KUKA KRL program: vw_hlf_usr_s.src, vw_hlf_usr_s.dat

--- vw_hlf_usr_s.src ---
&ACCESS RVEO
&REL 6
&COMMENT KS24.24.000_VW
&PARAM TPVW_VERSION = 8.1.8
&PARAM DISKPATH = VW_User / Applikation / VW_Grei_Fehl
DEF vw_hlf_usr_s( )
   ;
   ;*-----------------------------------------------------*
   ;* Erstellt am:                                        *
   ;* 2017.11.03                                          *
   ;*------------------------------------------------------
   ;
END
;
;FOLD INIT Handl_Fehl
GLOBAL DEF HLF_INIT( )
INT i
;;
;
END
;ENDFOLD
;
;-----------------------------------------------------------
;FOLD SAW Handl_Fehl
GLOBAL DEF HLF_SAW( )
INT i
;
;
END
;ENDFOLD
;
;-----------------------------------------------------------
;FOLD RESET Handl_Fehl
GLOBAL DEF HLF_RESET( )
INT i
;
;
END
;ENDFOLD
;
;-----------------------------------------------------------
;FOLD CANCEL Handl_Fehl
GLOBAL DEF HLF_CANCEL( )
INT i
;
;
END
;ENDFOLD
;
;-----------------------------------------------------------
;FOLD LOOP Handl_Fehl
GLOBAL DEF HLF_LOOP( )
INT i, j, k
BOOL R_POS_ABFRA
BOOL V_POS_ABFRA


FOR i = 1 TO 22
;Schleifentest
    CONTINUE
	IF ($OUT[15]==TRUE) OR ($IN[15]==TRUE) THEN  ; Bei Grundstellung alle Greifer deaktivieren
	;Fehlermedungen OFF
	  HLF_SPGR_AKT[i]=FALSE
	  HLF_F_SPANNZ=0
	  HLF_A_BIS_H=0
      FEHLER_SPG=0
      FEHLER_GRU=0
	  FEHLER_TKO=0
	  HLF_KLEIN_A_B=0
	  CONTINUE
	  $OUT[HLF_BGE_V_R]=FALSE
	  CONTINUE
      $OUT[HLF_BGE_SP_A]=FALSE
		IF i <=15 THEN
	       HLF_BGEKONT[i]=FALSE
		ENDIF
	ENDIF
	;------------------------------------------------------------------
	k=1
	CONTINUE
    IF (HLF_SPGR_AKT[i]==TRUE) AND ($IN[15]==FALSE)  AND (HLF_OPT_SPS>=127) AND (HLF_OPT_SPS<=257) THEN  ;Spanngruppe aktiv
        ;-----Spanngruppe ist geschlossen--------------
    	IF (HLF_SPGR_AUF[I]==FALSE) THEN ; Spanngruppe ist geschlossen
	     FOR j = 1 TO (HLF_ANZ_SGRUP[i])  ; 2
		 ;----------Wechsel zwischen Abfrageposition
			IF (J==1) THEN
				R_POS_ABFRA=TRUE
				IF (HLF_ERSBIT_R[i]==TRUE) THEN  ; Erstes Bit ist R Pos
					R_POS_ABFRA=FALSE
				ENDIF
			ELSE
				IF (R_POS_ABFRA==FALSE) THEN
					R_POS_ABFRA=TRUE
				ELSE
					R_POS_ABFRA=FALSE
				ENDIF
			ENDIF
            ;-------ENDE---Wechsel zwischen Abfrageposition
          ;-----Kontrolle Spanngruppe--------------
			CONTINUE
         IF ( (HLF_ST_ADR_SG[i]+(j-1))<1) OR  ((HLF_ST_ADR_SG[i]+(j-1))> 4096) THEN
				HLF_ST_ADR_SG[i]=4070
			ENDIF
		    IF ($IN[(HLF_ST_ADR_SG[i]+(j-1))]<>R_POS_ABFRA) THEN ;; Kontrolle Position NIO
                IF (FEHLER_SPG<1) THEN
					;; FEHLERAUSGABE
					HLF_F_SPANNZ=i
					HLF_A_BIS_H=(j+1)/2
					HLF_KLEIN_A_B=0
					FEHLER_SPG=i
					FEHLER_GRU=j
					CONTINUE
					$OUT[HLF_BGE_V_R]= TRUE
					IF (i<17) THEN   ; Ausgabe Bit 11 Spanngruppe = True
						CONTINUE
					   $OUT[HLF_BGE_SP_A]=TRUE
					ELSE  ; Ausgabe Bit 11 Sauger = False
						CONTINUE
					   $OUT[HLF_BGE_SP_A]=FALSE
					   HLF_A_BIS_H=0
					ENDIF
				ENDIF
			ELSE
				IF (FEHLER_SPG>0) THEN  ; Fehler loeschen
					IF (FEHLER_SPG==i) AND (FEHLER_GRU==j) THEN
						HLF_F_SPANNZ=0
						HLF_A_BIS_H=0
						FEHLER_SPG=0
						FEHLER_GRU=0
						CONTINUE
						$OUT[HLF_BGE_V_R]=FALSE
						CONTINUE
						$OUT[HLF_BGE_SP_A]=FALSE
					ENDIF
				ENDIF
			ENDIF

		 ENDFOR
		 ;---ENDE--Spanngruppe ist geschlossen--------------
	   ELSE
	        ;---Start--Spanngruppe ist offen--------------
		FOR j = 1 TO (HLF_ANZ_SGRUP[i])
		    ;----------Wechsel zwischen Abfrageposition
			IF (J==1) THEN
				V_POS_ABFRA=FALSE
				IF (HLF_ERSBIT_R[i]==TRUE) THEN  ; Erstes Bit ist R Pos
					V_POS_ABFRA=TRUE
				ENDIF
			ELSE
				IF (V_POS_ABFRA==FALSE) THEN
					V_POS_ABFRA=TRUE
				ELSE
					V_POS_ABFRA=FALSE
				ENDIF
			ENDIF
            ;-------ENDE---Wechsel zwischen Abfrageposition
          ;-----Kontrolle Spanngruppe--------------

			CONTINUE
		    IF ($IN[(HLF_ST_ADR_SG[i]+(j-1))]<>V_POS_ABFRA) THEN ;; Kontrolle Position NIO
                IF (FEHLER_SPG<1) THEN
					;; FEHLERAUSGABE
					HLF_F_SPANNZ=i
					HLF_A_BIS_H=(j+1)/2
					HLF_KLEIN_A_B=0
					FEHLER_SPG=i
					FEHLER_GRU=j
					CONTINUE
					$OUT[HLF_BGE_V_R]= FALSE
					IF (i<17) THEN   ; Ausgabe Bit 11 Spanngruppe = True
						CONTINUE
					   $OUT[HLF_BGE_SP_A]=TRUE
					ELSE  ; Ausgabe Bit 11 Sauger = False
					   CONTINUE
					   $OUT[HLF_BGE_SP_A]=FALSE
					   HLF_A_BIS_H=0
					ENDIF
				ENDIF
			ELSE
				IF (FEHLER_SPG>0) THEN  ; Fehler loeschen
					IF (FEHLER_SPG==i) AND (FEHLER_GRU==j) THEN
						HLF_F_SPANNZ=0
						HLF_A_BIS_H=0
						FEHLER_SPG=0
						FEHLER_GRU=0
						CONTINUE
						$OUT[HLF_BGE_V_R]=FALSE
						CONTINUE
						$OUT[HLF_BGE_SP_A]=FALSE
					ENDIF
				ENDIF
			ENDIF

		 ENDFOR

			;---ENDE--Spanngruppe ist geschlossen--------------
	   ENDIF
    ELSE
	  IF (HLF_SPGR_AKT[i]==FALSE) AND (FEHLER_SPG==i) THEN
   	     HLF_F_SPANNZ=0
	     HLF_A_BIS_H=0
         FEHLER_SPG=0
         FEHLER_GRU=0
	     CONTINUE
		 $OUT[HLF_BGE_V_R]=FALSE
         CONTINUE
		 $OUT[HLF_BGE_SP_A]=FALSE
	  ENDIF

	ENDIF


;------------Teilkontrolle----------------

	CONTINUE
	If (i<=15) AND (HLF_F_SPANNZ<=0) AND ($IN[15]==FALSE) THEN ; Teilkontrollen
		IF (HLF_BGEKONT[i]==FALSE) AND (FEHLER_TKO==i) THEN ;FEHLER Ruecksetzen wenn nicht aktiv
			HLF_A_BIS_H=0
			FEHLER_TKO=0
			HLF_KLEIN_A_B=0
		ENDIF
		IF (HLF_BGEBITA[i]<1) OR (HLF_BGEBITA[i]>4096) THEN ; Fehlerabfang Abfrage Eingabe
         HLF_BGEBITA[i]=4070
		ENDIF
		IF (HLF_BGEBITB[i]<1) OR (HLF_BGEBITB[i]>4096) THEN  ; Fehlerabfang Abfrage Eingabe
         HLF_BGEBITB[i]=4070
		ENDIF
		IF (HLF_BGEKONT[i]==TRUE) AND ((FEHLER_TKO==i) OR (FEHLER_TKO<=0)) THEN   ;Bauteilkontrolle aktiv und (aktueller Fehler oder kein Fehler)
			IF (HLF_BGETEILV[i]==TRUE) THEN  ; Teilkontrolle Teil ist vorhanden
				CONTINUE
				IF (HLF_BGEMITAB[i]==TRUE) THEN  ;Mit klein A und B
					IF ($IN[(HLF_BGEBITA[i])]==TRUE) AND ($IN[(HLF_BGEBITB[i])]==TRUE) THEN ;; Bauteilkontrolle klein A Nicht vorhanden
						IF (FEHLER_TKO==i)  THEN ; Rücksetzen Fehler
							HLF_A_BIS_H=0
							FEHLER_TKO=0
							HLF_KLEIN_A_B=0
						ENDIF
					ELSE  ; FEHLERAUSGABE
						HLF_A_BIS_H=i
						FEHLER_TKO=i
						IF ($IN[(HLF_BGEBITA[i])]==FALSE) THEN
							HLF_KLEIN_A_B=1
						ELSE
							HLF_KLEIN_A_B=2
						ENDIF
					ENDIF

				ELSE   ; Ohne klein A und B
					IF ($IN[(HLF_BGEBITA[i])]==TRUE) THEN ;; Bauteilkontrolle klein A auf vorhanden
						IF (FEHLER_TKO==i)  THEN ; Rücksetzen Fehler
							HLF_A_BIS_H=0
							FEHLER_TKO=0
							HLF_KLEIN_A_B=0
						ENDIF
					ELSE  ; FEHLERAUSGABE
						HLF_A_BIS_H=i
						FEHLER_TKO=i
						HLF_KLEIN_A_B=0
					ENDIF
				ENDIF
			ELSE  ; Teilkontrolle Teil ist NICHT vorhanden

;------------     Auswertung Teilkontrolle KEIN Teil vorhanden
				IF (HLF_BGEMITAB[i]==TRUE) THEN  ;Mit klein A und B
					IF ($IN[(HLF_BGEBITA[i])]==FALSE) AND ($IN[(HLF_BGEBITB[i])]==FALSE) THEN ;; Bauteilkontrolle klein A Nicht vorhanden
						IF (FEHLER_TKO==i)  THEN ; Rücksetzen Fehler
							HLF_A_BIS_H=0
							FEHLER_TKO=0
							HLF_KLEIN_A_B=0
						ENDIF
					ELSE  ; FEHLERAUSGABE
						HLF_A_BIS_H=i
						FEHLER_TKO=i
						IF ($IN[(HLF_BGEBITA[i])]==TRUE) THEN
							HLF_KLEIN_A_B=1
						ELSE
							HLF_KLEIN_A_B=2
						ENDIF
					ENDIF

				ELSE   ; Ohne klein A und B

					IF ($IN[(HLF_BGEBITA[i])]==FALSE) THEN ;; Bauteilkontrolle klein A Nicht vorhanden
						IF (FEHLER_TKO==i)  THEN ; Rücksetzen Fehler
							HLF_A_BIS_H=0
							FEHLER_TKO=0
							HLF_KLEIN_A_B=0
						ENDIF
					ELSE  ; FEHLERAUSGABE
						HLF_A_BIS_H=i
						FEHLER_TKO=i
						HLF_KLEIN_A_B=0
					ENDIF

				ENDIF


			ENDIF ; Teilkontrolle Teil ist vorhanden ENDE
		ENDIF  ; Bauteilkontrolle ENDE
		;;;;; KLEIB b
    ;  ---------------------------

	ENDIF

	IF (HLF_OPT_SPS>127) THEN
		CONTINUE
		HLF_BIN5_AUS((HLF_OPT_SPS), HLF_F_SPANNZ) ; Ausgabe Spannzylinder
		CONTINUE
		HLF_BIN4_AUS((HLF_OPT_SPS+5), HLF_A_BIS_H) ; Ausgabe Teilkontrolle
		CONTINUE
		HLF_BIN2_AUS((HLF_OPT_SPS+11), HLF_KLEIN_A_B) ; Ausgabe Klein A_B
	ENDIF
ENDFOR
;
END
;ENDFOLD

;FOLD Werteausgabe 4 BIT
DEF HLF_BIN4_AUS(HLF_STARTADD :IN, HLF_WERT :IN)
INT HLF_STARTADD, HLF_WERT
IF (HLF_STARTADD>0) AND (HLF_STARTADD<500) AND (HLF_WERT<17) AND (HLF_WERT>=0) THEN

	IF (HLF_WERT>=8) THEN
		HLF_WERT = (HLF_WERT-8)
		CONTINUE
		$OUT[HLF_STARTADD+3]=TRUE
	ELSE
		CONTINUE
		$OUT[HLF_STARTADD+3]=FALSE
	ENDIF

	IF (HLF_WERT>=4) THEN
		HLF_WERT = (HLF_WERT-4)
		CONTINUE
		$OUT[(HLF_STARTADD+2)]=TRUE
	ELSE
		CONTINUE
		$OUT[(HLF_STARTADD+2)]=FALSE
	ENDIF

	IF (HLF_WERT>=2) THEN
		HLF_WERT = (HLF_WERT-2)
		CONTINUE
		$OUT[(HLF_STARTADD+1)]=TRUE
	ELSE
		CONTINUE
		$OUT[(HLF_STARTADD+1)]=FALSE
	ENDIF

		IF (HLF_WERT>=1) THEN
		HLF_WERT = (HLF_WERT-1)
		CONTINUE
		$OUT[(HLF_STARTADD)]=TRUE
	ELSE
		CONTINUE
		$OUT[(HLF_STARTADD)]=FALSE
	ENDIF


ENDIF

END
;ENDFOLD

;FOLD Werteausgabe 5 BIT
DEF HLF_BIN5_AUS(HLF_STARTADD :IN, HLF_WERT :IN)
INT HLF_STARTADD, HLF_WERT
IF (HLF_STARTADD>0) AND (HLF_STARTADD<500) AND (HLF_WERT<33) AND (HLF_WERT>=0) AND (HLF_OPT_SPS>127) THEN

	IF (HLF_WERT>=16) THEN
		HLF_WERT = (HLF_WERT-16)
		CONTINUE
		$OUT[HLF_STARTADD+4]=TRUE
	ELSE
		CONTINUE
		$OUT[HLF_STARTADD+4]=FALSE
	ENDIF

	IF (HLF_WERT>=8) THEN
		HLF_WERT = (HLF_WERT-8)
		CONTINUE
		$OUT[HLF_STARTADD+3]=TRUE
	ELSE
		CONTINUE
		$OUT[HLF_STARTADD+3]=FALSE
	ENDIF

	IF (HLF_WERT>=4) THEN
		HLF_WERT = (HLF_WERT-4)
		CONTINUE
		$OUT[(HLF_STARTADD+2)]=TRUE
	ELSE
		CONTINUE
		$OUT[(HLF_STARTADD+2)]=FALSE
	ENDIF

	IF (HLF_WERT>=2) THEN
		HLF_WERT = (HLF_WERT-2)
		CONTINUE
		$OUT[(HLF_STARTADD+1)]=TRUE
	ELSE
		CONTINUE
		$OUT[(HLF_STARTADD+1)]=FALSE
	ENDIF

		IF (HLF_WERT>=1) THEN
		HLF_WERT = (HLF_WERT-1)
		CONTINUE
		$OUT[(HLF_STARTADD)]=TRUE
	ELSE
		CONTINUE
		$OUT[(HLF_STARTADD)]=FALSE
	ENDIF

ENDIF

END
;ENDFOLD

;FOLD Werteausgabe 2 BIT
DEF HLF_BIN2_AUS(HLF_STARTADD :IN, HLF_WERT :IN)
INT HLF_STARTADD, HLF_WERT
IF (HLF_STARTADD>0) AND (HLF_STARTADD<500) AND(HLF_WERT<4) AND (HLF_WERT>=0) AND (HLF_OPT_SPS>127) THEN


	IF (HLF_WERT>=2) THEN
		HLF_WERT = (HLF_WERT-2)
		CONTINUE
		$OUT[(HLF_STARTADD+1)]=TRUE
	ELSE
		CONTINUE
		$OUT[(HLF_STARTADD+1)]=FALSE
	ENDIF

		IF (HLF_WERT>=1) THEN
		HLF_WERT = (HLF_WERT-1)
		CONTINUE
		$OUT[(HLF_STARTADD)]=TRUE
	ELSE
		CONTINUE
		$OUT[(HLF_STARTADD)]=FALSE
	ENDIF


ENDIF

END
;ENDFOLD

--- vw_hlf_usr_s.dat ---
&ACCESS  RV
&COMMENT KS24.24.000_VW
&PARAM DISKPATH = VW_User/Applikation/VW_GREI_FEHL
&PARAM TPVW_VERSION = 8.1.8
&REL 6
DEFDAT  vw_hlf_usr_s PUBLIC
;
;*-----------------------------------------------------*
;* Erstellt am:                                        *
;* 2017.11.03                                          *
;*------------------------------------------------------
;
;
GLOBAL BOOL HLF_IAKTIV=FALSE
GLOBAL BOOL Mit_HLF=FALSE

GLOBAL INT FEHLER_SPG=0
GLOBAL INT FEHLER_GRU=0
GLOBAL INT FEHLER_TKO=0
GLOBAL INT FEHLER_TKB=0

;FOLD Handl_Fehl Version1
GLOBAL INT HLF_STARTADR=0
GLOBAL INT HLF_SP_END=0
GLOBAL INT HLF_ABISH_ST=0
GLOBAL INT HLF_ABISH_EN=0
GLOBAL INT HLF_FEHLERTY=0

GLOBAL INT HLF_OPT_SPS=0


GLOBAL INT HLF_F_SPANNZ=0 ;Fehlerausgabe Spannzylinder
GLOBAL INT HLF_A_BIS_H=0 ;Fehlerausgabe A_bis_H
GLOBAL INT HLF_BGE_V_R=0
GLOBAL INT HLF_BGE_SP_A=0
GLOBAL INT HLF_KLEIN_A_B=0

GLOBAL INT HLF_MAX_SPA_G=22
GLOBAL BOOL HLF_FEHLER_E=FALSE

;Parameter
GLOBAL INT HLF_USR_PARA[6]
HLF_USR_PARA[1]=0
HLF_USR_PARA[2]=0
HLF_USR_PARA[3]=0
HLF_USR_PARA[4]=0
HLF_USR_PARA[5]=0
HLF_USR_PARA[6]=0

GLOBAL BOOL HLF_SPGR_AKT[22]
; Greifer Ueberwachung Spanngruppe N ist aktiv
HLF_SPGR_AKT[1]=FALSE
HLF_SPGR_AKT[2]=FALSE
HLF_SPGR_AKT[3]=FALSE
HLF_SPGR_AKT[4]=FALSE
HLF_SPGR_AKT[5]=FALSE
HLF_SPGR_AKT[6]=FALSE
HLF_SPGR_AKT[7]=FALSE
HLF_SPGR_AKT[8]=FALSE
HLF_SPGR_AKT[9]=FALSE
HLF_SPGR_AKT[10]=FALSE
HLF_SPGR_AKT[11]=FALSE
HLF_SPGR_AKT[12]=FALSE
HLF_SPGR_AKT[13]=FALSE
HLF_SPGR_AKT[14]=FALSE
HLF_SPGR_AKT[15]=FALSE
HLF_SPGR_AKT[16]=FALSE
;Sauger ab 17
HLF_SPGR_AKT[17]=FALSE
HLF_SPGR_AKT[18]=FALSE
HLF_SPGR_AKT[19]=FALSE
HLF_SPGR_AKT[20]=FALSE
HLF_SPGR_AKT[21]=FALSE
HLF_SPGR_AKT[22]=FALSE

;Stellungsmerker Greifer ist AUF und elektrisch in R
GLOBAL BOOL HLF_SPGR_AUF[22]
HLF_SPGR_AUF[1]=FALSE
HLF_SPGR_AUF[2]=FALSE
HLF_SPGR_AUF[3]=FALSE
HLF_SPGR_AUF[4]=FALSE
HLF_SPGR_AUF[5]=FALSE
HLF_SPGR_AUF[6]=FALSE
HLF_SPGR_AUF[7]=FALSE
HLF_SPGR_AUF[8]=FALSE
HLF_SPGR_AUF[9]=FALSE
HLF_SPGR_AUF[10]=FALSE
HLF_SPGR_AUF[11]=FALSE
HLF_SPGR_AUF[12]=FALSE
HLF_SPGR_AUF[13]=FALSE
HLF_SPGR_AUF[14]=FALSE
HLF_SPGR_AUF[15]=FALSE
HLF_SPGR_AUF[16]=FALSE
;Sauger ab 17
HLF_SPGR_AUF[17]=FALSE
HLF_SPGR_AUF[18]=FALSE
HLF_SPGR_AUF[19]=FALSE
HLF_SPGR_AUF[20]=FALSE
HLF_SPGR_AUF[21]=FALSE
HLF_SPGR_AUF[22]=FALSE

; Greifer Teilkontrolle erstes Bit oder klein a
GLOBAL INT HLF_BGEBITA[22]
HLF_BGEBITA[1]=4070
HLF_BGEBITA[2]=4070
HLF_BGEBITA[3]=4070
HLF_BGEBITA[4]=4070
HLF_BGEBITA[5]=4070
HLF_BGEBITA[6]=4070
HLF_BGEBITA[7]=4070
HLF_BGEBITA[8]=4070
HLF_BGEBITA[9]=4070
HLF_BGEBITA[10]=4070
HLF_BGEBITA[11]=4070
HLF_BGEBITA[12]=4070
HLF_BGEBITA[13]=4070
HLF_BGEBITA[14]=4070
HLF_BGEBITA[15]=4070
HLF_BGEBITA[16]=-1
HLF_BGEBITA[17]=-1
HLF_BGEBITA[18]=-1
HLF_BGEBITA[19]=-1
HLF_BGEBITA[20]=-1
HLF_BGEBITA[21]=-1
HLF_BGEBITA[22]=-1

; Greifer Teilkontrolle, zweites BIT (klein b)
GLOBAL INT HLF_BGEBITB[22]
HLF_BGEBITB[1]=4070
HLF_BGEBITB[2]=4070
HLF_BGEBITB[3]=4070
HLF_BGEBITB[4]=4070
HLF_BGEBITB[5]=4070
HLF_BGEBITB[6]=4070
HLF_BGEBITB[7]=4070
HLF_BGEBITB[8]=4070
HLF_BGEBITB[9]=4070
HLF_BGEBITB[10]=4070
HLF_BGEBITB[11]=4070
HLF_BGEBITB[12]=4070
HLF_BGEBITB[13]=4070
HLF_BGEBITB[14]=4070
HLF_BGEBITB[15]=4070
HLF_BGEBITB[16]=-1
HLF_BGEBITB[17]=-1
HLF_BGEBITB[18]=-1
HLF_BGEBITB[19]=-1
HLF_BGEBITB[20]=-1
HLF_BGEBITB[21]=-1
HLF_BGEBITB[22]=-1

GLOBAL BOOL HLF_BGEMITAB[22]
; Auswahl Greifer Teilkontrolle mit klein a und b
HLF_BGEMITAB[1]=FALSE
HLF_BGEMITAB[2]=FALSE
HLF_BGEMITAB[3]=FALSE
HLF_BGEMITAB[4]=FALSE
HLF_BGEMITAB[5]=FALSE
HLF_BGEMITAB[6]=FALSE
HLF_BGEMITAB[7]=FALSE
HLF_BGEMITAB[8]=FALSE
HLF_BGEMITAB[9]=FALSE
HLF_BGEMITAB[10]=FALSE
HLF_BGEMITAB[11]=FALSE
HLF_BGEMITAB[12]=FALSE
HLF_BGEMITAB[13]=FALSE
HLF_BGEMITAB[14]=FALSE
HLF_BGEMITAB[15]=FALSE
HLF_BGEMITAB[16]=FALSE
HLF_BGEMITAB[17]=FALSE
HLF_BGEMITAB[18]=FALSE
HLF_BGEMITAB[19]=FALSE
HLF_BGEMITAB[20]=FALSE
HLF_BGEMITAB[21]=FALSE
HLF_BGEMITAB[22]=FALSE

GLOBAL BOOL HLF_BGETEILV[22]
; Greifer Teilkontrolle, Teil ist vorhanden
HLF_BGETEILV[1]=FALSE
HLF_BGETEILV[2]=FALSE
HLF_BGETEILV[3]=FALSE
HLF_BGETEILV[4]=FALSE
HLF_BGETEILV[5]=FALSE
HLF_BGETEILV[6]=FALSE
HLF_BGETEILV[7]=FALSE
HLF_BGETEILV[8]=FALSE
HLF_BGETEILV[9]=FALSE
HLF_BGETEILV[10]=FALSE
HLF_BGETEILV[11]=FALSE
HLF_BGETEILV[12]=FALSE
HLF_BGETEILV[13]=FALSE
HLF_BGETEILV[14]=FALSE
HLF_BGETEILV[15]=FALSE
HLF_BGETEILV[16]=FALSE
HLF_BGETEILV[17]=FALSE
HLF_BGETEILV[18]=FALSE
HLF_BGETEILV[19]=FALSE
HLF_BGETEILV[20]=FALSE
HLF_BGETEILV[21]=FALSE
HLF_BGETEILV[22]=FALSE

GLOBAL BOOL HLF_BGEKONT[22]
; Greifer Teilkontrolle aktiv schalten
HLF_BGEKONT[1]=FALSE
HLF_BGEKONT[2]=FALSE
HLF_BGEKONT[3]=FALSE
HLF_BGEKONT[4]=FALSE
HLF_BGEKONT[5]=FALSE
HLF_BGEKONT[6]=FALSE
HLF_BGEKONT[7]=FALSE
HLF_BGEKONT[8]=FALSE
HLF_BGEKONT[9]=FALSE
HLF_BGEKONT[10]=FALSE
HLF_BGEKONT[11]=FALSE
HLF_BGEKONT[12]=FALSE
HLF_BGEKONT[13]=FALSE
HLF_BGEKONT[14]=FALSE
HLF_BGEKONT[15]=FALSE
HLF_BGEKONT[16]=FALSE
HLF_BGEKONT[17]=FALSE
HLF_BGEKONT[18]=FALSE
HLF_BGEKONT[19]=FALSE
HLF_BGEKONT[20]=FALSE
HLF_BGEKONT[21]=FALSE
HLF_BGEKONT[22]=FALSE

;Startadresse Greifer Spanner Eingaben
GLOBAL INT HLF_ST_ADR_SG[22]
HLF_ST_ADR_SG[1]=-1
HLF_ST_ADR_SG[2]=-1
HLF_ST_ADR_SG[3]=-1
HLF_ST_ADR_SG[4]=-1
HLF_ST_ADR_SG[5]=-1
HLF_ST_ADR_SG[6]=-1
HLF_ST_ADR_SG[7]=-1
HLF_ST_ADR_SG[8]=-1
HLF_ST_ADR_SG[9]=-1
HLF_ST_ADR_SG[10]=-1
HLF_ST_ADR_SG[11]=-1
HLF_ST_ADR_SG[12]=-1
HLF_ST_ADR_SG[13]=-1
HLF_ST_ADR_SG[14]=-1
HLF_ST_ADR_SG[15]=-1
HLF_ST_ADR_SG[16]=-1
;Sauger
HLF_ST_ADR_SG[17]=-1
HLF_ST_ADR_SG[18]=-1
HLF_ST_ADR_SG[19]=-1
HLF_ST_ADR_SG[20]=-1
HLF_ST_ADR_SG[21]=-1
HLF_ST_ADR_SG[22]=-1

;Anzahl der Bits der Eingaben je Spanngruppe
GLOBAL INT HLF_ANZ_SGRUP[22]
HLF_ANZ_SGRUP[1]=-1
HLF_ANZ_SGRUP[2]=-1
HLF_ANZ_SGRUP[3]=-1
HLF_ANZ_SGRUP[4]=-1
HLF_ANZ_SGRUP[5]=-1
HLF_ANZ_SGRUP[6]=-1
HLF_ANZ_SGRUP[7]=-1
HLF_ANZ_SGRUP[8]=-1
HLF_ANZ_SGRUP[9]=-1
HLF_ANZ_SGRUP[10]=-1
HLF_ANZ_SGRUP[11]=-1
HLF_ANZ_SGRUP[12]=-1
HLF_ANZ_SGRUP[13]=-1
HLF_ANZ_SGRUP[14]=-1
HLF_ANZ_SGRUP[15]=-1
HLF_ANZ_SGRUP[16]=-1
;Sauger ab 17
HLF_ANZ_SGRUP[17]=-1
HLF_ANZ_SGRUP[18]=-1
HLF_ANZ_SGRUP[19]=-1
HLF_ANZ_SGRUP[20]=-1
HLF_ANZ_SGRUP[21]=-1
HLF_ANZ_SGRUP[22]=-1

; Greifer erstes Bit ist Rueck Pos
GLOBAL BOOL HLF_ERSBIT_R[22]
HLF_ERSBIT_R[1]=TRUE
HLF_ERSBIT_R[2]=TRUE
HLF_ERSBIT_R[3]=TRUE
HLF_ERSBIT_R[4]=TRUE
HLF_ERSBIT_R[5]=TRUE
HLF_ERSBIT_R[6]=TRUE
HLF_ERSBIT_R[7]=TRUE
HLF_ERSBIT_R[8]=TRUE
HLF_ERSBIT_R[9]=TRUE
HLF_ERSBIT_R[10]=TRUE
HLF_ERSBIT_R[11]=TRUE
HLF_ERSBIT_R[12]=TRUE
HLF_ERSBIT_R[13]=TRUE
HLF_ERSBIT_R[14]=TRUE
HLF_ERSBIT_R[15]=TRUE
HLF_ERSBIT_R[16]=TRUE
;Sauger ab 17
HLF_ERSBIT_R[17]=FALSE
HLF_ERSBIT_R[18]=TRUE
HLF_ERSBIT_R[19]=TRUE
HLF_ERSBIT_R[20]=TRUE
HLF_ERSBIT_R[21]=TRUE
HLF_ERSBIT_R[22]=TRUE

;; ----------------------------------------
;ENDFOLD

ENDDAT
